TYPE ST_DB_Enthalpie_r134a :
STRUCT
	id: DINT;
	timestamp: DT;
	Temperatur: STRING(45);
	h1: STRING(45);
	h1_5: STRING(45);
	h2: STRING(45);
	h2_5: STRING(45);
	h3: STRING(45);
	h3_5: STRING(45);
	h4: STRING(45);
	h4_5: STRING(45);
	h5: STRING(45);
	h5_5: STRING(45);
	h6: STRING(45);
	h6_5: STRING(45);
	h7: STRING(45);
	h7_5: STRING(45);
	h8: STRING(45);
	h8_5: STRING(45);
	h9: STRING(45);
	h9_5: STRING(45);
	h10: STRING(45);
	h10_5: STRING(45);
	h11: STRING(45);
	h11_5: STRING(45);
	h12: STRING(45);
	h12_5: STRING(45);
	h13: STRING(45);
	h13_5: STRING(45);
	h14: STRING(45);
	h14_5: STRING(45);
	h15: STRING(45);
END_STRUCT
END_TYPE

(* stored: Version 1.1.0.1, ProductVersion 3.1.4019.2
   DUT ST_DB_Enthalpie_r134a: Id {b7cfdc55-d8e3-4fdc-b195-2d229dc523db} *)
